// TIA Portal V17 export
// export: Created 2022-07-20T06:59:48.4823097Z, ExportSetting WithDefaults, DisplayName Totally Integrated Automation Portal, DisplayVersion V17, DisplayName TIA Portal Openness, DisplayVersion V17, DisplayName TIA Portal Version Control Interface, DisplayVersion V17, DisplayName SINAMICS Startdrive Advanced, DisplayVersion V17, DisplayName SINAMICS Startdrive G130, G150, S120, S150, SINAMICS MV, S210, DisplayVersion V17, DisplayName SINAMICS Startdrive G110M, G120, G120C, G120D, G120P, G115D, DisplayVersion V17, DisplayName STEP 7 Professional, DisplayVersion V17, DisplayName STEP 7 Safety, DisplayVersion V17, DisplayName WinCC Advanced, DisplayVersion V17
FUNCTION_BLOCK "FB10201_SubomduleAlarmManagement"   // FB10201, LAD
{ S7_Optimized_Access := 'TRUE' }
VERSION : 0.1
// stored: AutoNumber false, IsIECCheckEnabled false, IsRetainMemResEnabled false, MemoryReserve 100, SetENOAutomatically false, UDAEnableTagReadback false
   VAR_INPUT
      Acknowledge { ExternalAccessible := 'False'; ExternalVisible := 'False'; ExternalWritable := 'False'} : Bool;
      DBName { ExternalAccessible := 'False'; ExternalVisible := 'False'; ExternalWritable := 'False'} : String;
   END_VAR
   VAR_IN_OUT
      MachineAlarms : "stStandardMgiMachineAlarms";
      SubmoduleAlarms : "stStandardMgiSubmoduleAlarms";
   END_VAR
   VAR
      R_TRIG_NewInfoAlarmDetected : R_TRIG;
   END_VAR
   VAR_TEMP
      i : SInt;
      SubmoduleAlarms_INFO_Temp : DWord;
      i_string : String;
   END_VAR
BEGIN

REGION Network 1 (SCL): Edge Signals & Timers
   REGION EDGE SIGNALS
       #R_TRIG_NewInfoAlarmDetected(CLK := #SubmoduleAlarms.INFO <> #SubmoduleAlarms_INFO_Temp);
   END_REGION
END_REGION

REGION Network 2 (SCL): Acknowledge Management
   IF #Acknowledge THEN
       #SubmoduleAlarms.ESTOP := 16#0;
       #MachineAlarms.ESTOP_Detected := #SubmoduleAlarms.ESTOP_Detected := FALSE;

       #SubmoduleAlarms.STOP := 16#0;
       #MachineAlarms.STOP_Detected := #SubmoduleAlarms.STOP_Detected := FALSE;

       #SubmoduleAlarms.HOLD := 16#0;
       #MachineAlarms.HOLD_Detected := #SubmoduleAlarms.HOLD_Detected := FALSE;
   END_IF;

   IF #Acknowledge THEN
       #SubmoduleAlarms.INFO := 16#0;
       #MachineAlarms.INFO_Detected := #SubmoduleAlarms.INFO_Detected := FALSE;
       #SubmoduleAlarms_INFO_Temp := #SubmoduleAlarms.INFO; //Store The Info Alarm Temp After Resetting All Alarms
   END_IF;

   IF #R_TRIG_NewInfoAlarmDetected.Q THEN
       #SubmoduleAlarms_INFO_Temp := #SubmoduleAlarms.INFO; //Store The Info Alarm Temp Before Resetting All Alarms
       #SubmoduleAlarms.INFO := 16#0;
       #MachineAlarms.INFO_Detected := #SubmoduleAlarms.INFO_Detected := FALSE;
   END_IF;
END_REGION

REGION Network 3 (SCL): Estop Alarm Detection Management
   //Alarm Detection
   IF #SubmoduleAlarms.ESTOP <> 16#0 THEN
       #SubmoduleAlarms.ESTOP_Detected := TRUE;
       #MachineAlarms.ESTOP_Detected := TRUE;
   END_IF;

   (* //First Alarm Detection
   IF #SubmoduleAlarms.ESTOP_Detected AND #MachineAlarms.ESTOP_FirstAlarm = '' THEN
       #i := "FC10028_FirstBitActivatedInValue"(#SubmoduleAlarms.ESTOP);
       IF #SubmoduleAlarms.ESTOP_String[#i] = '' AND (LEN(#DBName) < 200) THEN
           #MachineAlarms.ESTOP_FirstAlarm := CONCAT(IN1 := #DBName, IN2 := '.Alarms.ESTOP[', IN3 := DELETE(IN := SINT_TO_STRING(#i), L := 1, P := 1), IN4 := ']');
       ELSIF #SubmoduleAlarms.ESTOP_String[#i] <> '' AND LEN(#SubmoduleAlarms.ESTOP_String[#i]) < 250 THEN
           #MachineAlarms.ESTOP_FirstAlarm := #SubmoduleAlarms.ESTOP_String[#i];
       ELSE
           #MachineAlarms.ESTOP_FirstAlarm := 'Estop Alarm Text Cannot Be Generated';
       END_IF;
   END_IF; *)

   //Splitting Dword To 2 Word For HMI
   "FC10332_DWordTo2Words"(DWord_Input:=#SubmoduleAlarms.ESTOP,
                           Word_HighWeight=>#SubmoduleAlarms.ESTOP_HMI[1],
                           Word_LowWeight=>#SubmoduleAlarms.ESTOP_HMI[0]);
END_REGION

REGION Network 4 (SCL): Stop Alarm Detection Management
   //Alarm Detection
   IF #SubmoduleAlarms.STOP <> 16#0 THEN
       #SubmoduleAlarms.STOP_Detected := TRUE;
       #MachineAlarms.STOP_Detected := TRUE;
   END_IF;

   (* //First Alarm Detection
   IF #SubmoduleAlarms.STOP_Detected AND #MachineAlarms.STOP_FirstAlarm = '' THEN
       #i := "FC10028_FirstBitActivatedInValue"(#SubmoduleAlarms.STOP);
       IF #SubmoduleAlarms.STOP_String[#i] = '' AND (LEN(#DBName) < 200) THEN
           #MachineAlarms.STOP_FirstAlarm := CONCAT(IN1 := #DBName, IN2 := '.Alarms.STOP[', IN3 := DELETE(IN := SINT_TO_STRING(#i), L := 1, P := 1), IN4 := ']');
       ELSIF #SubmoduleAlarms.STOP_String[#i] <> '' AND LEN(#SubmoduleAlarms.STOP_String[#i]) < 250 THEN
           #MachineAlarms.STOP_FirstAlarm := #SubmoduleAlarms.STOP_String[#i];
       ELSE
           #MachineAlarms.STOP_FirstAlarm := 'Stop Alarm Text Cannot Be Generated';
       END_IF;
   END_IF; *)

   //Splitting Dword To 2 Word For HMI
   "FC10332_DWordTo2Words"(DWord_Input := #SubmoduleAlarms.STOP,
                           Word_HighWeight => #SubmoduleAlarms.STOP_HMI[1],
                           Word_LowWeight => #SubmoduleAlarms.STOP_HMI[0]);
END_REGION

REGION Network 5 (SCL): Hold Alarm Detection Management
   //Alarm Detection
   IF #SubmoduleAlarms.HOLD <> 16#0 THEN
       #SubmoduleAlarms.HOLD_Detected := TRUE;
       #MachineAlarms.HOLD_Detected := TRUE;
   END_IF;

   (* //First Alarm Detection
   IF #SubmoduleAlarms.HOLD_Detected AND #MachineAlarms.HOLD_FirstAlarm = '' THEN
       #i := "FC10028_FirstBitActivatedInValue"(#SubmoduleAlarms.HOLD);
       IF #SubmoduleAlarms.HOLD_String[#i] = '' AND (LEN(#DBName) < 200) THEN
           #MachineAlarms.HOLD_FirstAlarm := CONCAT(IN1 := #DBName, IN2 := '.Alarms.HOLD[', IN3 := DELETE(IN := SINT_TO_STRING(#i), L := 1, P := 1), IN4 := ']');
       ELSIF #SubmoduleAlarms.HOLD_String[#i] <> '' AND LEN(#SubmoduleAlarms.HOLD_String[#i]) < 250 THEN
           #MachineAlarms.HOLD_FirstAlarm := #SubmoduleAlarms.HOLD_String[#i];
       ELSE
           #MachineAlarms.HOLD_FirstAlarm := 'Hold Alarm Text Cannot Be Generated';
       END_IF;
   END_IF; *)

   //Splitting Dword To 2 Word For HMI
   "FC10332_DWordTo2Words"(DWord_Input := #SubmoduleAlarms.HOLD,
                           Word_HighWeight => #SubmoduleAlarms.HOLD_HMI[1],
                           Word_LowWeight => #SubmoduleAlarms.HOLD_HMI[0]);
END_REGION

REGION Network 6 (SCL): Info Alarm Detection Management
   //Alarm Detection
   IF #SubmoduleAlarms.INFO <> 16#0 THEN
       #SubmoduleAlarms.INFO_Detected := TRUE;
       #MachineAlarms.INFO_Detected := TRUE;
   END_IF;

   (* //First Alarm Detection
   IF #SubmoduleAlarms.INFO_Detected AND #MachineAlarms.INFO_FirstAlarm = '' THEN
       #i := "FC10028_FirstBitActivatedInValue"(#SubmoduleAlarms.INFO);
       IF #SubmoduleAlarms.INFO_String[#i] = '' AND (LEN(#DBName) < 200) THEN
           #MachineAlarms.INFO_FirstAlarm := CONCAT(IN1 := #DBName, IN2 := '.Alarms.INFO[', IN3 := DELETE(IN := SINT_TO_STRING(#i), L := 1, P := 1), IN4 := ']');
       ELSIF #SubmoduleAlarms.INFO_String[#i] <> '' AND LEN(#SubmoduleAlarms.INFO_String[#i]) < 250 THEN
           #MachineAlarms.INFO_FirstAlarm := #SubmoduleAlarms.INFO_String[#i];
       ELSE
           #MachineAlarms.INFO_FirstAlarm := 'Info Alarm Text Cannot Be Generated';
       END_IF;
   END_IF; *)

   //Splitting Dword To 2 Word For HMI
   "FC10332_DWordTo2Words"(DWord_Input := #SubmoduleAlarms.HOLD,
                           Word_HighWeight => #SubmoduleAlarms.INFO_HMI[1],
                           Word_LowWeight => #SubmoduleAlarms.INFO_HMI[0]);
END_REGION
END_FUNCTION_BLOCK
